FUNCTION_BLOCK FB_Conveyor IMPLEMENTS I_actuator
VAR
    bEnabled : BOOL;
    bRunning : BOOL;
	bDisabled : BOOL;
END_VAR

METHOD Disable : bool
VAR_INPUT
END_VAR
bEnabled := FALSE;
END_METHOD

METHOD Enable : bool
VAR_INPUT
END_VAR
bEnabled := TRUE;
END_METHOD

METHOD Init : bool
VAR_INPUT
END_VAR
bEnabled := FALSE;
bRunning := FALSE;
END_METHOD

METHOD Start : bool
VAR_INPUT
END_VAR
IF bEnabled THEN
    bRunning := TRUE;
END_IF
END_METHOD

METHOD Stop : bool
VAR_INPUT
END_VAR
bEnabled := FALSE;
END_METHOD

METHOD Update : bool
VAR_INPUT
END_VAR
IF NOT bEnabled THEN
    bRunning := FALSE;
END_IF
END_METHOD

END_FUNCTION_BLOCK

(* stored: Version 1.1.0.1
   POU FB_Conveyor: Id {e00c0afe-0881-4a47-afe2-90d576be7e63}, SpecialFunc None
   Method Disable: Id {6e586afe-8ebe-4907-a3db-d639603c3eea}
   Method Enable: Id {5893a5f0-da79-4b0b-82b7-1d272ee67f61}
   Method Init: Id {330c59b6-b0a2-4d14-8ff5-66341457b5bf}
   Method Start: Id {fb0a2b4f-c51a-4b67-8b87-ddedd7c020db}
   Method Stop: Id {791c2abf-0ecb-4492-a591-d7b52ea55ce4}
   Method Update: Id {faf0b631-5f22-4c95-bee6-01bd10fabeaa} *)
